// TIA Portal V19 export
TYPE "LEXCHANGETRAY_typeAxisSimpleControlNode_2"
// stored: Access Published
   STRUCT
      commandConfiguration : "LEXCHANGETRAY_typeAxisSimpleControlCommandConfiguration2";
      commands : "LEXCHANGETRAY_typeAxisSimpleControlNodeCommands_2";
      monitoring : "LEXCHANGETRAY_typeAxisSimpleControlNodeMonitoring_2";
   END_STRUCT;
END_TYPE
